// TIA Portal V18 export
TYPE "ProcessData"
// stored: IsFailsafeCompliant false
   STRUCT
      PartStatus : Int;   // 产品状态
      PartSNGCode : Int;   // 产品NG代码
      PartRemoveFlag : Bool;
      Spare1 : Bool;
      Spare2 : Bool;
      Spare3 : Bool;
      Spare4 : Bool;
      Spare5 : Bool;
      Spare6 : Bool;
      Spare7 : Bool;
      Spare8 : Bool;
      Spare9 : Bool;
      Spare10 : Bool;
      Spare11 : Bool;
      Spare12 : Bool;
      Spare13 : Bool;
      Spare14 : Bool;
      Spare15 : Bool;
      ShaftCode { S7_SetPoint := 'True'} : String[128];   // 轴条码
      RingCode_1 { S7_SetPoint := 'True'} : String[128];   // 条码
      Code_1 : String[128];
      RingCode_2 : String[128];
      TableCode_1 : String[128];
      TableCode_2 : String[128];
      Press1Program : Int;
      Press1FinalPosition : Real;
      Press1FinalForce : Real;
      Press2Program : Int;
      Press2FinalPosition : Real;
      Press2FinalForce : Real;
      IV3_ShaftCheckResult : Int;
      IV3_ShaftScore_1 : Int;
      IV3_ShaftScore_2 : Int;
      IV3_ShaftScore_3 : Int;
      IV3_ShaftScore_4 : Int;
      IV3_MagnetCheckResult : Int;
      IV3_MagnetScore : Int;
      Spare_3 : Array[0..89] of Int;
   END_STRUCT;
END_TYPE
